Fanuc KAREL source: kt00297.KL

-- PROVISIONAL review KL for V1013-1; original PC SHA256 4b5fb789781214a3bbe278b4aadbb130c5181ee712ce67e726b632949a9e23a2
-- Incomplete behavior may be omitted. Consult companion uncertainty JSON. Do not deploy.
PROGRAM KT00297
%NOLOCKGROUP
VAR
  R1 : REAL
  I2 : INTEGER
  OUT : BOOLEAN
BEGIN
  -- UNRESOLVED_PC offsets 5-16; opcodes 2E,23
  -- UNRESOLVED_PC offsets 21-32; opcodes 2E,23
  -- UNRESOLVED_PC offsets 37-57; opcodes 21,21,64,6E,23
  -- UNRESOLVED_PC offsets 62-66; opcodes 7F
END KT00297
